VAR_GLOBAL CONSTANT
	MAX_EC_SLAVES : UINT := 49;
END_VAR

(* stored: Version 1.1.0.1, ProductVersion 3.1.4026.18
   GVL EtherCatParameter: Id {3c947b34-68f8-4997-8ab5-70b51281d5e8}, ParameterList True *)
